PROGRAM FAST
VAR
	nChan : INT;
	MOS_TS: INT;
	i: INT;	
	ChannelMHTFunction : ARRAY[0..MAX_USED_CHANNEL_IDX] OF HLI3_QuitChannelMHTFunction;
END_VAR

(****************************************************************************************)
(*	  							Wait for HLI initialization								*)
(****************************************************************************************)
IF NOT CNCSystem.bHLIInit THEN
	RETURN;
END_IF

IF PRG_CNCChannelHandler.stOptions.bDisableMFunctHandling THEN
	FOR i := 0 TO MAX_USED_CHANNEL_IDX DO
		ChannelMHTFunction[i](nChanIdx:=0, bM30Acknowledgement := TRUE);
	END_FOR
END_IF	

(* Programm call for MOS_TS M functions *)
// PRG_FastMFunctions();

END_PROGRAM

(* stored: Version 1.1.0.1, ProductVersion 3.1.4024.9
   POU FAST: Id {16c202d0-b697-4d74-8856-0055624c8fd5}, SpecialFunc None *)
